(*
DESCRIPTION: This function block is responsible for printing the results of the tests to a defined output.
*)
FUNCTION_BLOCK FB_MessagePrinter

METHOD PUBLIC LogMessageError
VAR_INPUT
    sExpected : STRING;
    sActual : STRING;
    sMessage : Tc2_System.T_MaxString;
    sTestInstancePath : Tc2_System.T_MaxString;
END_VAR
VAR
    sTestInstancePathCleaned : STRING;
    sFinalMessage : Tc2_System.T_MaxString;
END_VAR
sTestInstancePathCleaned := RemoveInstancePathAndProjectNameFromTestInstancePath(sTestInstancePath);
sFinalMessage := Tc2_Standard.CONCAT('FAILED TEST $'', sTestInstancePathCleaned);
sFinalMessage := Tc2_Standard.CONCAT(sFinalMessage, '$'');
IF Tc2_Standard.LEN(STR := sExpected) > 0 THEN
    sFinalMessage := Tc2_Standard.CONCAT(sFinalMessage, ', EXP: ');
    sFinalMessage := Tc2_Standard.CONCAT(sFinalMessage, sExpected);
END_IF
IF Tc2_Standard.LEN(STR := sActual) > 0 THEN
    sFinalMessage := Tc2_Standard.CONCAT(sFinalMessage, ', ACT: ');
    sFinalMessage := Tc2_Standard.CONCAT(sFinalMessage, sActual);
END_IF
IF Tc2_Standard.LEN(STR := sMessage) > 0 THEN
    sFinalMessage := Tc2_Standard.CONCAT(sFinalMessage, ', MSG: %s ');
END_IF
Tc2_System.ADSLOGSTR(msgCtrlMask := Tc2_System.ADSLOG_MSGTYPE_ERROR,
                     msgFmtStr := sFinalMessage,
                     strArg := sMessage);
END_METHOD

METHOD PRIVATE RemoveInstancePathAndProjectNameFromTestInstancePath : STRING
VAR_INPUT
    sTestInstancePath : Tc2_System.T_MaxString;
END_VAR
VAR
    nCharacterPositionOfProjectName : INT;
    sProjectNameWithDot : STRING;
END_VAR
// Add the '.' character to the project name for search
sProjectNameWithDot := CONCAT(STR1 := TwinCAT_SystemInfoVarList._AppInfo.ProjectName, STR2 := '.');

// Find the character position of the beginning of the first occurence of the project name
nCharacterPositionOfProjectName := FIND(sTestInstancePath, sProjectNameWithDot);


IF nCharacterPositionOfProjectName > 0 THEN
    sTestInstancePath := DELETE(STR := sTestInstancePath,
                                LEN := LEN(sProjectNameWithDot),
                                POS := nCharacterPositionOfProjectName);
END_IF

// Check if the project name happens to be the same as namespace, and in that case, remove that as well
nCharacterPositionOfProjectName := FIND(sTestInstancePath,
                                        sProjectNameWithDot);

IF nCharacterPositionOfProjectName > 0 THEN
    sTestInstancePath := DELETE(STR := sTestInstancePath,
                                LEN := LEN(sProjectNameWithDot),
                                POS := nCharacterPositionOfProjectName);
END_IF

RemoveInstancePathAndProjectNameFromTestInstancePath := sTestInstancePath;
END_METHOD

END_FUNCTION_BLOCK

(* stored: Version 1.1.0.1, ProductVersion 3.1.4022.12
   POU FB_MessagePrinter: Id {54911d7d-b4a4-43a8-a981-a2fc14a13f71}, SpecialFunc None
   Method LogMessageError: Id {bab195d7-5e96-4c3f-8266-c59551de8d0d}
   Method RemoveInstancePathAndProjectNameFromTestInstancePath: Id {60392e51-c21c-4caa-851a-442a6a14bf1d} *)
